// TIA Portal V19 export
FUNCTION "HMI_Call" : Void   // FC12, LAD
// stored: SetENOAutomatically false
BEGIN

REGION Network 1
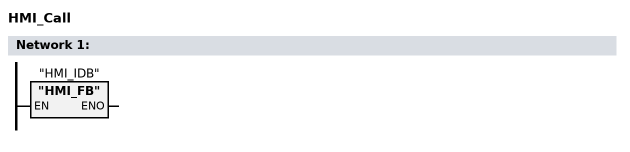
   RUNG wire#powerrail
      "HMI_IDB"()
   END_RUNG
   // the same network as SCL:
   "HMI_IDB"();   // "HMI_FB"
END_REGION
END_FUNCTION
